// 电机控制主逻辑
IF Stop THEN
  Running := FALSE;
  CurrentState := 0;
  ActualSpeed := 0;
ELSIF Start THEN
  Running := TRUE;
  CurrentState := 1;
  
  // 速度斜坡调节
  IF ActualSpeed < SpeedSetpoint THEN
    ActualSpeed := ActualSpeed + SpeedRampStep;
    IF ActualSpeed > SpeedSetpoint THEN
      ActualSpeed := SpeedSetpoint;
    END_IF;
  ELSIF ActualSpeed > SpeedSetpoint THEN
    ActualSpeed := ActualSpeed - SpeedRampStep;
    IF ActualSpeed < SpeedSetpoint THEN
      ActualSpeed := SpeedSetpoint;
    END_IF;
  END_IF;
ELSE
  // 保持当前状态
  IF CurrentState = 1 THEN
    Running := TRUE;
    // 保持当前速度
  ELSE
    Running := FALSE;
    ActualSpeed := 0;
  END_IF;
END_IF;
